Fanuc KAREL source: KT00276.KL

PROGRAM KT00276
%NOLOCKGROUP
VAR
  P1: POSITION
  P2: XYZWPR
  OUT: BOOLEAN
BEGIN
    P2.Y = 2.0
  OUT = P1 = P2
END KT00276
